FUNCTION_BLOCK AGVEvaluate (* Tamplate for a simple Basic Function Block Type *)
  (* Standard: 61499-2 *)
  (* Version 0.0, 2018-03-27, 4DIAC-IDE, 4DIAC-Consortium *)
  (* Version 1.0, 2016-05-26, AZ, fortiss GmbH *)
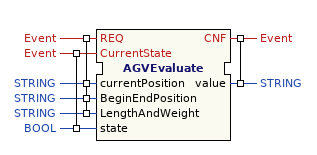
  EVENT_INPUT
    REQ WITH currentPosition, BeginEndPosition, LengthAndWeight; (* Normal Execution Request *)
    CurrentState WITH state; (* idel or busy *)
  END_EVENT
  EVENT_OUTPUT
    CNF WITH value; (* Execution Confirmation *)
  END_EVENT
  VAR_INPUT
    currentPosition : STRING;
    BeginEndPosition : STRING; (* like 1_10 *)
    LengthAndWeight : STRING;
    state : BOOL;
  END_VAR
  VAR_OUTPUT
    value : STRING;
  END_VAR
  VAR
    currentTime : DINT; (* Internal Variable *)
    LastTime : DINT; (* Internal Variable *)
  END_VAR
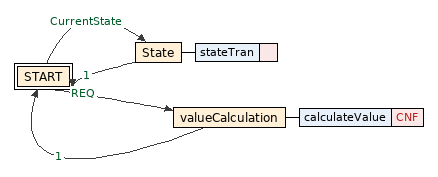
  EC_STATES
    START; (* Initial State *)
    State : stateTran;
    valueCalculation : calculateValue -> CNF;
  END_STATES
  EC_TRANSITIONS
    START TO State := CurrentState;
    State TO START := 1;
    START TO valueCalculation := REQ;
    valueCalculation TO START := 1;
  END_TRANSITIONS
  ALGORITHM stateTran IN ST: (* new algorithm *)

  END_ALGORITHM
  ALGORITHM calculateValue IN ST: (* new algorithm *)

  END_ALGORITHM
END_FUNCTION_BLOCK
